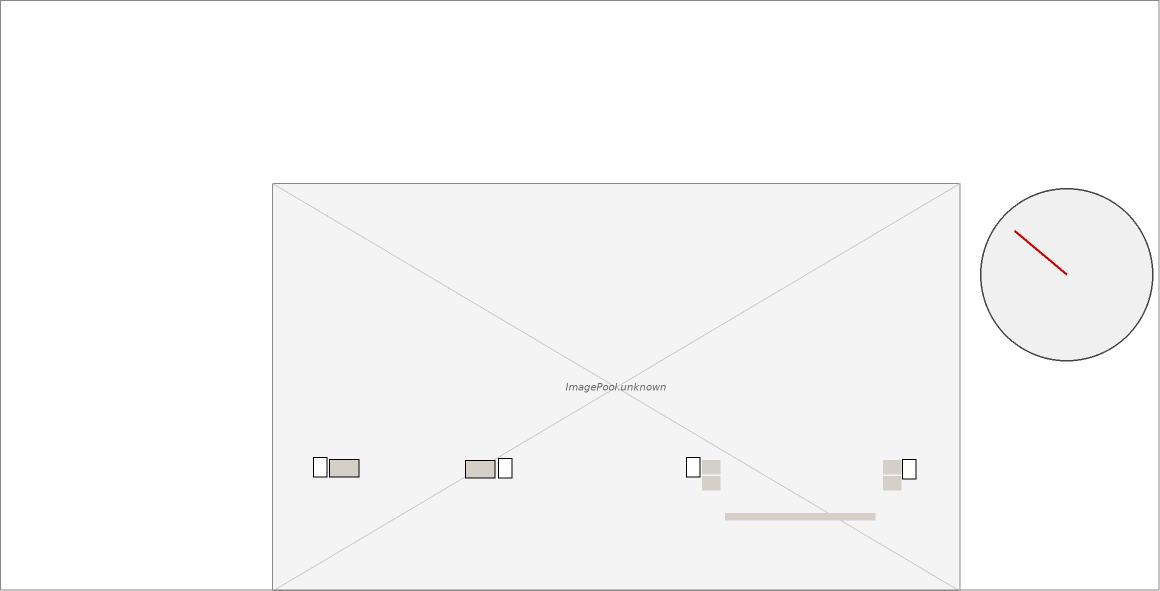
VISUALIZATION testLights  // 1160x591
    Image (272,183 688x408), image: ImagePool.unknown
    RoundedRectangle (498,458 14x20), colour toggle: GVL_Lights.BlinkerLeft
    RoundedRectangle (313,457 14x20), colour toggle: GVL_Lights.BlinkerRight
    RoundedRectangle (465,460 30x18), colour toggle: GVL_Lights.LightsFront
    RoundedRectangle (686,457 14x20), colour toggle: GVL_Lights.BlinkerLeft
    RoundedRectangle (902,459 14x20), colour toggle: GVL_Lights.BlinkerRight
    RoundedRectangle (329,459 30x18), colour toggle: GVL_Lights.LightsFront
    RoundedRectangle (702,460 18x14), colour toggle: GVL_Lights.LightsRear
    RoundedRectangle (702,476 18x14), colour toggle: GVL_Lights.LightsBrake
    RoundedRectangle (883,460 18x14), colour toggle: GVL_Lights.LightsRear
    RoundedRectangle (883,476 18x14), colour toggle: GVL_Lights.LightsBrake
    RoundedRectangle (725,513 150x7), colour toggle: GVL_Lights.LightsReverse
    Meter90 (973,188 187x173), value: movements.PositionToDegree_0.Deg, style: Meter-Meter90-Gray, scale format: %.1f, scale -45..45
END_VISUALIZATION

(* stored: Version 1.1.0.1, ProductVersion 3.1.4024.3
   Visu testLights: Id {6bbcc6ff-faec-4775-90aa-a71f1d4f3c3c} *)
